FUNCTION_BLOCK EcMasterGetAbnortalStateChange IMPLEMENTS IEcTask
VAR_INPUT
END_VAR
VAR_OUTPUT
END_VAR
VAR
	iState : INT;
	masterAbnormalStateChanges : Tc2_EtherCAT.FB_EcGetAllSlaveAbnormalStateChanges;
	_abnormalStates : ARRAY[0..Tc2_EtherCAT.EC_MAX_SLAVES] OF UDINT;
	_execute: BOOL;
	_done: BOOL;
	_busy: BOOL;
	_error: BOOL;
	_netId: AMSNETID;
END_VAR

CASE iState OF
	0:
		IF _execute THEN
			_done := FALSE;
			_busy := TRUE;
			_error := FALSE;
			masterAbnormalStateChanges.bExecute := TRUE;
			IF masterAbnormalStateChanges.bBusy THEN
				iState := 10;
				_execute := false;
			END_IF
		END_IF
	10:
		IF NOT masterAbnormalStateChanges.bBusy THEN
			IF NOT masterAbnormalStateChanges.bError THEN
				_done := TRUE;
			ELSE
				_error := TRUE;
			END_IF
			_busy := FALSE;
			masterAbnormalStateChanges.bExecute := FALSE;
			iState := 0;
		END_IF
END_CASE

masterAbnormalStateChanges(sNetId := Tc2_System.F_CreateAmsNetId(nIds := NetId),
							pAddrBuf := ADR(_abnormalStates),
							cbBufLen := SIZEOF(_abnormalStates));

PROPERTY AbnormalStateChanges : reference to array[0..EC_MAX_Slaves] of udint
GET
AbnormalStateChanges REF= _abnormalStates;
END_GET
END_PROPERTY

{warning 'add method implementation '}
METHOD Abort : BOOL
masterAbnormalStateChanges.bExecute := FALSE;
_busy := FALSE;
_execute := FALSE;
Abort := TRUE;
iState := 0;
END_METHOD

{warning 'add property implementation'}
PROPERTY Busy : BOOL
GET
Busy := _busy;
END_GET
END_PROPERTY

{warning 'add property implementation'}
PROPERTY Done : BOOL
GET
Done := _done;
END_GET
END_PROPERTY

{warning 'add property implementation'}
PROPERTY Error : BOOL
GET
Error := _error;
END_GET
END_PROPERTY

{warning 'add method implementation '}
METHOD Execute : BOOL
IF NOT masterAbnormalStateChanges.bBusy THEN
	Execute := _execute := true;
END_IF
END_METHOD

{warning 'add property implementation'}
PROPERTY NetID : amsnetid
GET
NetID := _netId;
END_GET
SET
_netId := NetID;
END_SET
END_PROPERTY

END_FUNCTION_BLOCK

(* stored: Version 1.1.0.1, ProductVersion 3.1.4024.9
   POU EcMasterGetAbnortalStateChange: Id {dc855736-7955-4698-83a6-3179b98a1beb}, SpecialFunc None
   Property AbnormalStateChanges: Id {3dc925b7-38da-4eb9-bcb4-4e0648d5ab10}
   Get Get: Id {fb5f8561-4e5a-4cdd-a5df-4dbbc2c815d0}
   Method Abort: Id {7349edae-dc7e-4b83-8079-263014c9bca9}
   Property Busy: Id {e7541636-b459-4f78-9f19-9d241e4b0b2c}
   Get Get: Id {6b23289d-18f2-43d1-9342-09374770d2a5}
   Property Done: Id {57e58e3e-e07d-4a5d-a150-aeb5624e915e}
   Get Get: Id {f94572c6-08ca-4b59-859e-6724f684e217}
   Property Error: Id {2fdcee5d-203b-4558-b284-4f6ae7af1724}
   Get Get: Id {fdbda515-a579-4f80-89ce-82a6d595029a}
   Method Execute: Id {3fe26c6c-3187-404a-b668-73217a30a2cc}
   Property NetID: Id {d1a19152-0747-4b7b-8e1d-caae46b2a492}
   Get Get: Id {1c6c259b-241a-4e76-866e-a1ddd8987343}
   Set Set: Id {04f0557b-c4b3-410d-ab3e-6de24515810f} *)
